(* IEC 61131-3 sources: moqui-plc/iec61131/moqui/runtime/component/mantle-hvac/src/main/org/moqui/util/json, 4 files *)

(* ---- JsonToParametersMapper.pou ---- *)
(*#-#-#-#-#-#-#-#-#-#---Declaration---#-#-#-#-#-#-#-#-#-#-#-#-#*)

{attribute 'no_assign'}
FUNCTION_BLOCK JsonToParametersMapper
VAR_EXTERNAL
	dev : DeviceFacade;
END_VAR
VAR_INPUT
    jsonKey : WSTRING(255) := "";
    jsonValue : JSON.JSONElement;
END_VAR

(*#-#-#-#-#-#-#-#-#-#---Implementation---#-#-#-#-#-#-#-#-#-#-#-#-#*)

(* Args validation *)
IF (jsonKey = "") THEN RETURN; END_IF;

(* Mapping JSON elements to parameters, ignoring nknown keys and errors (non-blocking). *)
IF jsonKey = "tempSetpoint" THEN
    dev.tempSetpoint := TO_REAL(jsonValue.value.lrValue);
ELSIF jsonKey = "tempHysteresis" THEN
    dev.tempHysteresis := TO_REAL(jsonValue.value.lrValue);
ELSIF jsonKey = "coldGlycolEnableRequest" THEN
    dev.coldGroupEnableRequest := jsonValue.value.xValue;
ELSIF jsonKey = "workEffort.workEffortName" THEN
    workEffort.workEffortName := LEFT(TO_STRING(jsonValue.value.wsValue), 255);
	(* etc. *)
END_IF;

(* ---- JsonToParametersMapper.st ---- *)
FUNCTION_BLOCK JsonToParametersMapper
	VAR_EXTERNAL
		dev : DeviceFacade;
	END_VAR
	VAR_INPUT
	    jsonKey : WSTRING(255) := "";
	    jsonValue : JSON.JSONElement;
	END_VAR

	(* Args validation *)
	IF (jsonKey = "") THEN RETURN; END_IF;

	(* Mapping JSON elements to parameters, ignoring unknown keys and errors (non-blocking). *)

	(* --- 6-DOF robot arm trajectory (moqui-device export#Trajectory) ---
	 * JSON payload shape (received on MqttParameterSub topic, e.g. moqui/robot/arm1/trajectory):
	 *   { "approximatedFunctionId": "100051", "waypointCount": 10,
	 *     "axes": { "J1": [θ0,θ1,…,θ9], "J2": […], …, "J6": […] } }
	 *
	 * Each axis key ("J1"…"J6") carries a JSON array of REAL values (radians, sequenceNum order).
	 * The current FB handles only scalar values (jsonValue.value.lrValue).
	 * When implemented, each array branch would iterate jsonValue.elements and populate
	 * the application-specific trajectory buffer, e.g.:
	 *
	 *   ELSIF jsonKey = "J1" THEN
	 *       FOR i := 0 TO MIN(jsonValue.count - 1, MAX_WAYPOINTS - 1) DO
	 *           dev.trajectory.joint[0, i] := TO_LREAL(jsonValue.elements[i].value.lrValue);
	 *       END_FOR;
	 *   ELSIF jsonKey = "J2" THEN ...
	 *   (* J3→joint[2,i], J4→joint[3,i], J5→joint[4,i], J6→joint[5,i] *)
	 *
	 * In simatic-ax the target struct is Trajectory / TrajectoryPoint (see Trajectory.st).
	 * In Codesys adapt to the application DeviceFacade trajectory buffer.
	 *)

	IF jsonKey = "tempSetpoint" THEN
	    dev.tempSetpoint := TO_REAL(jsonValue.value.lrValue);
	ELSIF jsonKey = "tempHysteresis" THEN
	    dev.tempHysteresis := TO_REAL(jsonValue.value.lrValue);
	ELSIF jsonKey = "coldGlycolEnableRequest" THEN
	    dev.coldGroupEnableRequest := jsonValue.value.xValue;
	ELSIF jsonKey = "workEffort.workEffortName" THEN
	    workEffort.workEffortName := LEFT(TO_STRING(jsonValue.value.wsValue), 255);
		(* etc. *)
	END_IF;
	END_FUNCTION_BLOCK

(* ---- ParametersToJsonMapper.pou ---- *)
(*#-#-#-#-#-#-#-#-#-#---Declaration---#-#-#-#-#-#-#-#-#-#-#-#-#*)

{attribute 'no_assign'}
FUNCTION_BLOCK ParametersToJsonMapper
VAR_EXTERNAL
	dev : DeviceFacade;
END_VAR
VAR_IN_OUT
    jsonBuilder : JSON.JSONBuilder;
END_VAR
VAR_INPUT
    rootIndex : DINT;
END_VAR

(*#-#-#-#-#-#-#-#-#-#---Implementation---#-#-#-#-#-#-#-#-#-#-#-#-#*)

(* Mapping parameters to JSON elements, ignoring errors *)
jsonBuilder.SetKeyWithValue("processActualDuration", dev.processActualDuration, rootIndex);
jsonBuilder.SetKeyWithValue("actualRuntime", dev.actualRuntime, rootIndex);
jsonBuilder.SetKeyWithValue("actualBreakDuration", dev.actualBreakDuration, rootIndex);
jsonBuilder.SetKeyWithValue("airFlowActuatorFault", dev.airFlow.actuatorFault, rootIndex);
(* etc. *)

(* ---- ParametersToJsonMapper.st ---- *)
FUNCTION_BLOCK ParametersToJsonMapper
	VAR_EXTERNAL
		dev : DeviceFacade;
	END_VAR
	VAR_IN_OUT
	    jsonBuilder : JSON.JSONBuilder;
	END_VAR
	VAR_INPUT
	    rootIndex : DINT;
	END_VAR

	(* Approved HVAC live-parameter surface. Keep keys aligned with
	 * HVACDemoData.xml DeviceRequestItem.requestItemName values. *)
	jsonBuilder.SetKeyWithValue("tempSetpoint", dev.tempSetpoint, rootIndex);
	jsonBuilder.SetKeyWithValue("tempHysteresis", dev.tempHysteresis, rootIndex);
	jsonBuilder.SetKeyWithValue("tempMin", dev.tempMin, rootIndex);
	jsonBuilder.SetKeyWithValue("tempMax", dev.tempMax, rootIndex);
	jsonBuilder.SetKeyWithValue("rhSetpoint", dev.rhSetpoint, rootIndex);
	jsonBuilder.SetKeyWithValue("rhHysteresis", dev.rhHysteresis, rootIndex);
	jsonBuilder.SetKeyWithValue("rhMin", dev.rhMin, rootIndex);
	jsonBuilder.SetKeyWithValue("rhMax", dev.rhMax, rootIndex);
	jsonBuilder.SetKeyWithValue("ductTempMin", dev.ductTempMin, rootIndex);
	jsonBuilder.SetKeyWithValue("ductTempMax", dev.ductTempMax, rootIndex);
	jsonBuilder.SetKeyWithValue("ductRhMax", dev.ductRhMax, rootIndex);
	jsonBuilder.SetKeyWithValue("setPointTimeHigh", dev.setPointTimeHigh, rootIndex);
	jsonBuilder.SetKeyWithValue("setPointTimeLow", dev.setPointTimeLow, rootIndex);
	jsonBuilder.SetKeyWithValue("processEstimatedDuration", dev.processEstimatedDuration, rootIndex);
	jsonBuilder.SetKeyWithValue("processMinDuration", dev.processMinDuration, rootIndex);
	jsonBuilder.SetKeyWithValue("processRemainingDuration", dev.processRemainingDuration, rootIndex);
	jsonBuilder.SetKeyWithValue("estimatedRuntime", dev.estimatedRuntime, rootIndex);
	jsonBuilder.SetKeyWithValue("minRuntime", dev.minRuntime, rootIndex);
	jsonBuilder.SetKeyWithValue("estimatedBreakDuration", dev.estimatedBreakDuration, rootIndex);
	jsonBuilder.SetKeyWithValue("minBreakDuration", dev.minBreakDuration, rootIndex);

	(* Runtime telemetry is published alongside the configurable live surface. *)
	jsonBuilder.SetKeyWithValue("processActualDuration", dev.processActualDuration, rootIndex);
	jsonBuilder.SetKeyWithValue("actualRuntime", dev.actualRuntime, rootIndex);
	jsonBuilder.SetKeyWithValue("actualBreakDuration", dev.actualBreakDuration, rootIndex);
	jsonBuilder.SetKeyWithValue("airFlowActuatorFault", dev.airFlow.actuatorFault, rootIndex);
	END_FUNCTION_BLOCK
